PROGRAM HTTP_DEMO_1
VAR
	url_text : STRING := 'http://weather.yahooapis.com/forecastrss?p=94089&u=c';
	URL_DATA : URL;
	IP_C: IP_C;
	S_BUF: NETWORK_BUFFER;
	R_BUF: NETWORK_BUFFER;
	IP_CONTROL_1: IP_CONTROL;

	DNS_CLIENT: DNS_CLIENT;
	HTTP_GET: HTTP_GET;
	http_release: BOOL;
	enable: BOOL := TRUE;
	http_status: STRING;
	header_start: UINT;
	header_stop: UINT;
	body_start: UINT;
	body_stop: UINT;
	http_get_done: BOOL;
	http_get_error: DWORD;
	COUNT_DR: COUNT_DR;
	cycles: DWORD;
	TON_1: TON;
	F_TRIG: F_TRIG;
END_VAR
VAR // added by the converter: edge detectors and wires of the graphical bodies
    _w1 : ANY;
END_VAR

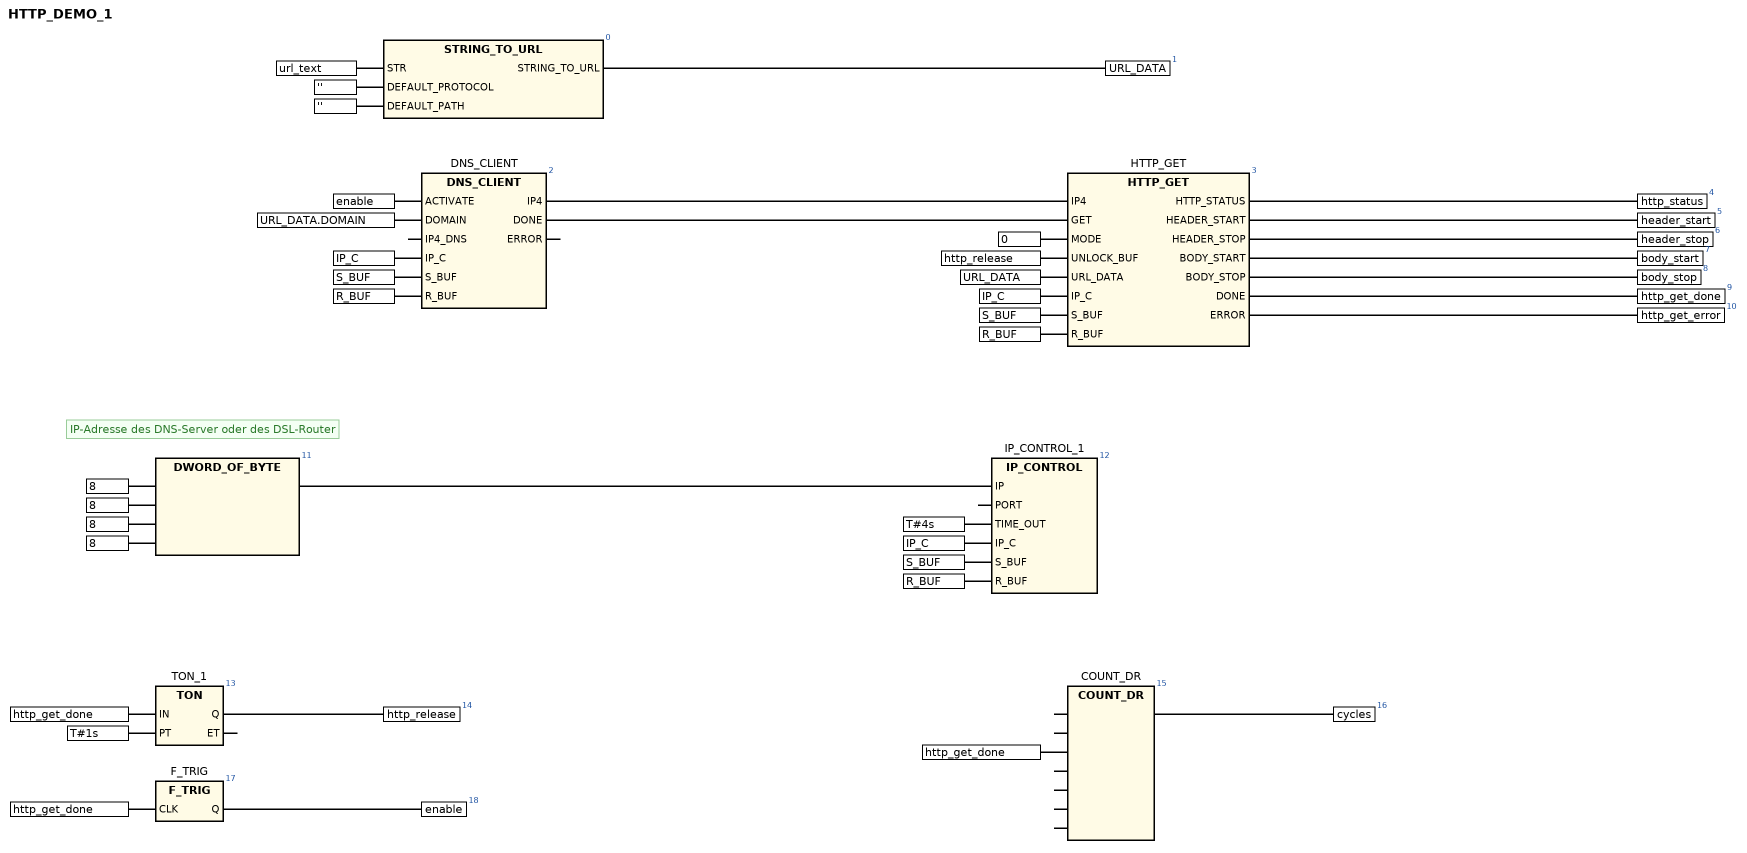
URL_DATA := STRING_TO_URL(STR := url_text, DEFAULT_PROTOCOL := '', DEFAULT_PATH := '');
DNS_CLIENT(ACTIVATE := enable, DOMAIN := URL_DATA.DOMAIN, IP_C := IP_C, S_BUF := S_BUF, R_BUF := R_BUF);
HTTP_GET(
    IP4 := DNS_CLIENT.IP4,
    GET := DNS_CLIENT.DONE,
    MODE := 0,
    UNLOCK_BUF := http_release,
    URL_DATA := URL_DATA,
    IP_C := IP_C,
    S_BUF := S_BUF,
    R_BUF := R_BUF);
http_status := HTTP_GET.HTTP_STATUS;
header_start := HTTP_GET.HEADER_START;
header_stop := HTTP_GET.HEADER_STOP;
body_start := HTTP_GET.BODY_START;
body_stop := HTTP_GET.BODY_STOP;
http_get_done := HTTP_GET.DONE;
http_get_error := HTTP_GET.ERROR;
// IP-Adresse des DNS-Server oder des DSL-Router
_w1 := DWORD_OF_BYTE(8, 8, 8, 8);
IP_CONTROL_1(IP := _w1, TIME_OUT := T#4s, IP_C := IP_C, S_BUF := S_BUF, R_BUF := R_BUF); // IP_CONTROL
TON_1(IN := http_get_done, PT := T#1s); // TON
http_release := TON_1.Q;
COUNT_DR(_in3 := http_get_done);
cycles := COUNT_DR._out1;
F_TRIG(CLK := http_get_done);
enable := F_TRIG.Q;

END_PROGRAM

(* stored: Version 1.1.0.1, ProductVersion 3.1.4024.0
   POU HTTP_DEMO_1: Id {c443e366-40d3-44db-be12-6f2ff7510d7d}, SpecialFunc None *)
